// TIA Portal V17 export
// export: Created 2022-07-20T07:01:28.0294157Z, ExportSetting WithDefaults, DisplayName Totally Integrated Automation Portal, DisplayVersion V17, DisplayName TIA Portal Openness, DisplayVersion V17, DisplayName TIA Portal Version Control Interface, DisplayVersion V17, DisplayName SINAMICS Startdrive Advanced, DisplayVersion V17, DisplayName SINAMICS Startdrive G130, G150, S120, S150, SINAMICS MV, S210, DisplayVersion V17, DisplayName SINAMICS Startdrive G110M, G120, G120C, G120D, G120P, G115D, DisplayVersion V17, DisplayName STEP 7 Professional, DisplayVersion V17, DisplayName STEP 7 Safety, DisplayVersion V17, DisplayName WinCC Advanced, DisplayVersion V17
FUNCTION_BLOCK "FB10180_ChucksManager"   // FB10180, LAD
{ S7_Optimized_Access := 'TRUE' }
VERSION : 0.1
// stored: AutoNumber false, IsIECCheckEnabled false, IsRetainMemResEnabled false, MemoryReserve 100, SetENOAutomatically false, UDAEnableTagReadback false
   VAR_INPUT
      ChucksCommunicationIn : Array[0..15] of "stChuckCommunicationIn";
      ChucksParameters : Array[0..15] of "stChuckParameters";
      NumberOfChucks : USInt;
   END_VAR
   VAR_OUTPUT
      ChucksCommunicationOut : Array[0..15] of "stChuckCommunicationOut";
      ChucksSafetyFeedbackHighSignal : Bool;
      ChucksSafetyFeedbackLowSignal : Bool;
      ChucksStartElec : Bool;
      ChucksStopInProgress : Bool;
      ChucksNormalStopDone : Bool;
      ChucksQuickStopDone : Bool;
   END_VAR
   VAR_IN_OUT
      ChucksRequests : Array[0..15] of "stChuckRequests";
      RequestChucksStartElecPulse : Bool;
      RequestChucksStartElecLevel : Bool;
      RequestNormalStop : Bool;
      RequestQuickStop : Bool;
      RequestStartJog : Bool;
      RequestStopJog : Bool;
      ChucksStates : Array[0..15] of "stChuckStates";
   END_VAR
   VAR
      ChucksSameOmacMode : Bool;
      ChucksSameOmacState : Bool;
      ChucksSameMaintenanceFeedback : Bool;
      i : USInt;
      JogManagementStateDiagram : Int;
      R_TRIG_ChucksRequest { S7_SetPoint := 'True'} : R_TRIG;
      R_TRIG_RequestAcknowledge { S7_SetPoint := 'True'} : R_TRIG;
      R_TRIG_ChucksStartElecPulse { S7_SetPoint := 'True'} : R_TRIG;
      R_TRIG_ChucksStartElecLevel { S7_SetPoint := 'True'} : R_TRIG;
      R_TRIG_ErrorOnChucks { S7_SetPoint := 'True'} : R_TRIG;
      R_TRIG_RequestStartJog { S7_SetPoint := 'True'} : R_TRIG;
      R_TRIG_RequestStopJog { S7_SetPoint := 'True'} : R_TRIG;
      F_TRIG_ChucksRequest { S7_SetPoint := 'True'} : F_TRIG;
      F_TRIG_ChucksStartElecLevel { S7_SetPoint := 'True'} : F_TRIG;
      TON_RequestDuration { S7_SetPoint := 'True'} : TON_TIME;
      TON_AcknowledgeDuration { S7_SetPoint := 'True'} : TON_TIME;
      TON_ChucksStartElecPulse { S7_SetPoint := 'True'} : TON_TIME;
      ArrayErrorsChucksLog : Array[0..15] of DInt;
      FB10182_ChuckPortionTracking_Instance { S7_SetPoint := 'True'} : Array[0..15] of "FB10182_ChuckPortionTracking";
   END_VAR
   VAR CONSTANT
      WAIT_FOR_JOG_REQUESTS : Int := 0;
      PARAMETER_CHUCKS : Int := 10;
      START_JOG : Int := 20;
      STOP_JOG : Int := 30;
      JOG_MANAGEMENT_DONE : Int := 40;
   END_VAR
BEGIN

REGION Network 1 (SCL): First Scan
   IF "FirstScan" THEN
       FOR #i := 0 TO #NumberOfChucks DO
           #ChucksCommunicationOut[#i].Acknowledge := FALSE;
           #ChucksCommunicationOut[#i].SheetManagement := 0;
           #ChucksCommunicationOut[#i].StartIdle := FALSE;
           #ChucksCommunicationOut[#i].StartInit := FALSE;
           #ChucksCommunicationOut[#i].Stop := FALSE;
       END_FOR;
       #ChucksCommunicationOut[0].MaintenanceFunction := 1;

       #JogManagementStateDiagram := #WAIT_FOR_JOG_REQUESTS;
   END_IF;
END_REGION

REGION Network 2 (SCL): Edge Signals & Timers
   REGION EDGE SIGNALS
       #R_TRIG_ChucksRequest(CLK := #ChucksRequests[0].StartInit OR #ChucksRequests[0].Stop OR #ChucksRequests[0].StartIdle);
       #R_TRIG_ChucksStartElecPulse(CLK := #RequestChucksStartElecPulse);
       #R_TRIG_ChucksStartElecLevel(CLK := #RequestChucksStartElecLevel);
       #R_TRIG_RequestAcknowledge(CLK := #ChucksRequests[0].Acknowledge);
       #R_TRIG_ErrorOnChucks(CLK := #ChucksStates[0].Error = -1);
       #R_TRIG_RequestStartJog(CLK := #RequestStartJog);
       #R_TRIG_RequestStopJog(CLK := #RequestStopJog);

       #F_TRIG_ChucksRequest(CLK := #ChucksRequests[0].StartInit OR #ChucksRequests[0].Stop OR #ChucksRequests[0].StartIdle);
       #F_TRIG_ChucksStartElecLevel(CLK := #RequestChucksStartElecLevel);
   END_REGION

   REGION TIMERS
       #TON_AcknowledgeDuration(IN := #ChucksCommunicationOut[0].Acknowledge,
                                PT := T#500ms);
       #TON_RequestDuration(IN := #ChucksRequests[0].StartInit OR #ChucksRequests[0].Stop OR #ChucksRequests[0].StartIdle,
                            PT := T#2s);
       #TON_ChucksStartElecPulse(IN := #RequestChucksStartElecPulse,
                                 PT := T#200ms);
   END_REGION
END_REGION

REGION Network 3 (SCL): Chucks Commands Management
   REGION START INIT / START IDLE / STOP / LOAD UNLOAD
       FOR #i := 0 TO #NumberOfChucks DO
           #ChucksCommunicationOut[#i].StartInit := #ChucksRequests[#i].StartInit;
           #ChucksCommunicationOut[#i].StartIdle := #ChucksRequests[#i].StartIdle;
           #ChucksCommunicationOut[#i].Stop := #ChucksRequests[#i].Stop;
           #ChucksCommunicationOut[#i].Load_Unload := #ChucksRequests[#i].Load_Unload;
           #ChucksCommunicationOut[#i].SheetManagement := #ChucksRequests[#i].SheetManagement;
       END_FOR;
   END_REGION

   REGION ACKNOWLEDGE
       IF #R_TRIG_RequestAcknowledge.Q THEN
           #ChucksCommunicationOut[0].Acknowledge := TRUE;
       ELSIF #TON_AcknowledgeDuration.Q THEN
           #ChucksCommunicationOut[0].Acknowledge := FALSE;
       END_IF;
   END_REGION

   REGION START ELEC
       //Start Elec Management
       IF #R_TRIG_ChucksStartElecLevel.Q OR #R_TRIG_ChucksStartElecPulse.Q THEN
           #ChucksStartElec := TRUE;
       ELSIF #TON_ChucksStartElecPulse.Q THEN
           #ChucksStartElec := FALSE;
       ELSIF #RequestNormalStop THEN
           IF #ChucksStates[#NumberOfChucks].ActualPosition > 23120.0 OR (#ChucksStates[#NumberOfChucks].ActualVelocity < 5.0 AND #ChucksStates[#NumberOfChucks / 2].ActualVelocity < 5.0) THEN
               #ChucksRequests[0].Stop := TRUE;
               #ChucksStartElec := FALSE;
           END_IF;
       ELSIF #RequestQuickStop THEN
           #ChucksRequests[0].Stop := TRUE;
           #ChucksStartElec := FALSE;
       ELSE
           #ChucksRequests[0].Stop := FALSE;
       END_IF;
   END_REGION

   REGION JOG
       IF #ChucksStates[0].Error <> 0 OR #R_TRIG_RequestStopJog.Q THEN
           #JogManagementStateDiagram := #STOP_JOG;
       END_IF;

       CASE #JogManagementStateDiagram OF
           #WAIT_FOR_JOG_REQUESTS:
               IF #ChucksStates[0].OmacState = "OMAC_STATE_STOPPED" AND #R_TRIG_RequestStartJog.Q THEN
                   #JogManagementStateDiagram := #PARAMETER_CHUCKS;
               END_IF;
           #PARAMETER_CHUCKS:
               //Request For Chucks
               #ChucksCommunicationOut[0].MaintenanceFunction := 2;

               //Condition To Go To Next Step
               IF #ChucksStates[0].MaintenanceFeedback = #ChucksCommunicationOut[0].MaintenanceFunction THEN
                   #JogManagementStateDiagram := #START_JOG;
               END_IF;
           #START_JOG:
               //Request For Chucks
               #ChucksRequests[0].StartInit := TRUE;

               //Condition To Go To Next Step
               IF #R_TRIG_RequestStopJog.Q THEN
                   #ChucksRequests[0].StartInit := FALSE;
                   #JogManagementStateDiagram := #STOP_JOG;
               END_IF;
           #STOP_JOG:
               #ChucksRequests[0].Stop := TRUE;
               #ChucksCommunicationOut[0].MaintenanceFunction := 1;

               IF #ChucksStates[0].OmacState = "OMAC_STATE_STOPPED" AND #ChucksStates[0].MaintenanceFeedback = 1 THEN
                   #ChucksRequests[0].Stop := FALSE;
                   #JogManagementStateDiagram := #JOG_MANAGEMENT_DONE;
               END_IF;
           #JOG_MANAGEMENT_DONE:
               #ChucksRequests[0].StartInit := FALSE;
               #ChucksRequests[0].Stop := FALSE;
               #JogManagementStateDiagram := #WAIT_FOR_JOG_REQUESTS;
       END_CASE;
   END_REGION

   REGION REQUEST PORTION TRACKING
       FOR #i := 1 TO #NumberOfChucks DO
           #ChucksRequests[#i].RequestPortionTracking := #ChucksRequests[0].RequestPortionTracking;
       END_FOR;
   END_REGION
END_REGION

REGION Network 4 (SCL): Chuck Potion Tracking Management
   FOR #i := 1 TO #NumberOfChucks DO
       #FB10182_ChuckPortionTracking_Instance[#i](EnablePortionTracking:=#ChucksRequests[#i].RequestPortionTracking,
                                                  StartPosition:=#ChucksParameters[#i].PortionTracking_StartDistance,
                                                  EndPosition:=#ChucksParameters[#i].PortionTracking_EndDistance,
                                                  ChuckActualPosition := #ChucksStates[#i].ActualPosition,
                                                  EndPositionReached=>#ChucksStates[#i].PortionTrackingDone);
   END_FOR;
END_REGION

REGION Network 5 (SCL): Chucks States Management
   #ChucksSameOmacMode := TRUE;
   #ChucksSafetyFeedbackHighSignal := FALSE;
   #ChucksSameOmacState := TRUE;
   #ChucksSameMaintenanceFeedback := TRUE;
   #ChucksStates[0].Enabled := TRUE;
   #ChucksStates[0].Initialized := TRUE;
   #ChucksStates[0].Prepositioned := TRUE;
   #ChucksStates[0].ChuckAlive := TRUE;
   #ChucksStates[0].OmacMode := 0;
   #ChucksStates[0].OmacState := 0;
   #ChucksStates[0].Error := 0;
   #ChucksStates[0].MaintenanceFeedback := 0;
   #ChucksStates[0].PortionTrackingDone := FALSE;
   #ChucksStates[0].SafetyFeedbackHighSignal := TRUE;
   #ChucksStates[0].SafetyFeedbackLowSignal := TRUE;

   IF #NumberOfChucks = 0 THEN
       #ChucksStates[0].Enabled := FALSE;
       #ChucksStates[0].Initialized := FALSE;
       #ChucksStates[0].Prepositioned := FALSE;
       #ChucksStates[0].SheetIn := FALSE;
       #ChucksStates[0].ChuckAlive := FALSE;
       #ChucksSameOmacMode := FALSE;
       #ChucksSameOmacState := FALSE;
       #ChucksStates[0].OmacMode := 0;
       #ChucksStates[0].OmacState := 0;
       #ChucksStates[0].Error := 0;
       #ChucksStates[0].MaintenanceFeedback := 0;
       #ChucksStates[0].PortionTrackingDone := FALSE;
   ELSIF #NumberOfChucks >= 1 THEN
       REGION CHUCKS STATES MANAGEMENT
           FOR #i := 1 TO #NumberOfChucks DO
               IF #ChucksStates[#i].ActualPosition < 0.0 THEN
                   #ChucksStates[#i].ActualPosition := 0.0;
               ELSIF #ChucksStates[#i].ActualPosition > 50000.0 THEN
                   #ChucksStates[#i].ActualPosition := 50000.0;
               ELSE
                   #ChucksStates[#i].ActualPosition := #ChucksCommunicationIn[#i].ActualPosition;
               END_IF;
               #ChucksStates[#i].ActualVelocity := #ChucksCommunicationIn[#i].ActualVelocity;
               #ChucksStates[#i].ChuckAlive := #ChucksCommunicationIn[#i].ChuckAlive;
               #ChucksStates[#i].Enabled := #ChucksCommunicationIn[#i].Enabled;
               #ChucksStates[#i].Error := #ChucksCommunicationIn[#i].Error;
               #ChucksStates[#i].Initialized := #ChucksCommunicationIn[#i].Initialized;
               #ChucksStates[#i].OmacMode := #ChucksCommunicationIn[#i].OmacMode;
               #ChucksStates[#i].OmacState := #ChucksCommunicationIn[#i].OmacState;
               #ChucksStates[#i].Prepositioned := #ChucksCommunicationIn[#i].Prepositioned;
               #ChucksStates[#i].SheetIn := #ChucksCommunicationIn[#i].SheetIn;
               #ChucksStates[#i].ChuckAlive := #ChucksCommunicationIn[#i].ChuckAlive;
               #ChucksStates[#i].MaintenanceFeedback := #ChucksCommunicationIn[#i].MaintenanceFeedback;
               #ChucksStates[#i].SafetyFeedbackHighSignal := #ChucksCommunicationIn[#i].ElectricalInputs.%X6;
               #ChucksStates[#i].SafetyFeedbackLowSignal := #ChucksCommunicationIn[#i].ElectricalInputs.%X6;
           END_FOR;
       END_REGION

       REGION DETERMINE COMMON STATE OF CHUCKS
           FOR #i := 1 TO #NumberOfChucks DO
               //Chucks Enabled States Management
               #ChucksStates[0].Enabled := #ChucksStates[0].Enabled AND #ChucksStates[#i].Enabled;

               //Chucks Initialzed States Management
               #ChucksStates[0].Initialized := #ChucksStates[0].Initialized AND #ChucksStates[#i].Initialized;

               //Chucks Prepositionned States Management
               #ChucksStates[0].Prepositioned := #ChucksStates[0].Prepositioned AND #ChucksStates[#i].Prepositioned;

               //Chucks Alive States Management
               #ChucksStates[0].ChuckAlive := #ChucksStates[0].ChuckAlive AND #ChucksStates[#i].ChuckAlive;

               //Chucks Safety Feedback Ok Management
               #ChucksStates[0].SafetyFeedbackHighSignal := #ChucksStates[0].SafetyFeedbackHighSignal AND #ChucksStates[#i].SafetyFeedbackHighSignal;

               //Chucks Safety Feedback Nok Management
               #ChucksStates[0].SafetyFeedbackLowSignal := #ChucksStates[0].SafetyFeedbackLowSignal AND NOT(#ChucksStates[#i].SafetyFeedbackLowSignal);
           END_FOR;
           #ChucksSafetyFeedbackHighSignal := #ChucksStates[0].SafetyFeedbackHighSignal;
           #ChucksSafetyFeedbackLowSignal := #ChucksStates[0].SafetyFeedbackLowSignal;

           //Chucks Sheet In Management
           FOR #i := 1 TO #NumberOfChucks DO
               IF #ChucksStates[#i].SheetIn THEN
                   #ChucksStates[0].SheetIn := TRUE;
                   EXIT;
               ELSE
                   #ChucksStates[0].SheetIn := FALSE;
               END_IF;
           END_FOR;

           //Chucks Error Management
           FOR #i := 1 TO #NumberOfChucks DO
               IF #ChucksStates[#i].Error <> 0 AND #ChucksStates[#i].Error <> 80000 THEN
                   #ChucksStates[0].Error := -1;
                   EXIT;
               ELSE
                   #ChucksStates[0].Error := 0;
               END_IF;
           END_FOR;

           //Chucks Omac Mode Management
           IF #NumberOfChucks = 1 THEN
               #ChucksStates[0].OmacMode := #ChucksStates[1].OmacMode;
           ELSIF #NumberOfChucks > 1 THEN
               FOR #i := 1 TO #NumberOfChucks - 1 DO
                   #ChucksSameOmacMode := #ChucksSameOmacMode AND (#ChucksStates[#i].OmacMode = #ChucksStates[#i + 1].OmacMode);
               END_FOR;
               IF #ChucksSameOmacMode THEN
                   #ChucksStates[0].OmacMode := #ChucksStates[1].OmacMode;
               ELSE
                   #ChucksStates[0].OmacMode := 0;
               END_IF;
           END_IF;

           //Chucks Omac State Management
           IF #NumberOfChucks = 1 THEN
               #ChucksStates[0].OmacState := #ChucksStates[1].OmacState;
           ELSIF #NumberOfChucks > 1 THEN
               FOR #i := 1 TO #NumberOfChucks - 1 DO
                   #ChucksSameOmacState := #ChucksSameOmacState AND (#ChucksStates[#i].OmacState = #ChucksStates[#i + 1].OmacState);
               END_FOR;
               IF #ChucksSameOmacState THEN
                   #ChucksStates[0].OmacState := #ChucksStates[1].OmacState;
               ELSE
                   #ChucksStates[0].OmacState := 0;
               END_IF;
           END_IF;

           //Chucks Maintenace Feedback Management
           IF #NumberOfChucks = 1 THEN
               #ChucksStates[0].MaintenanceFeedback := #ChucksStates[1].MaintenanceFeedback;
           ELSIF #NumberOfChucks > 1 THEN
               FOR #i := 1 TO #NumberOfChucks - 1 DO
                   #ChucksSameMaintenanceFeedback := #ChucksSameMaintenanceFeedback AND (#ChucksStates[#i].MaintenanceFeedback = #ChucksStates[#i + 1].MaintenanceFeedback);
               END_FOR;
               IF #ChucksSameMaintenanceFeedback THEN
                   #ChucksStates[0].MaintenanceFeedback := #ChucksStates[1].MaintenanceFeedback;
               ELSE
                   #ChucksStates[0].MaintenanceFeedback := 0;
               END_IF;
           END_IF;

           //Portion Tracking Done State Managment
           IF #NumberOfChucks = 1 THEN
               #ChucksStates[0].PortionTrackingDone := #ChucksStates[1].PortionTrackingDone;
           ELSIF #NumberOfChucks > 1 THEN
               FOR #i := 1 TO #NumberOfChucks - 1 DO
                   IF #ChucksStates[#i].PortionTrackingDone THEN
                       #ChucksStates[0].PortionTrackingDone := TRUE;
                       EXIT;
                   ELSE
                       #ChucksStates[0].PortionTrackingDone := FALSE;
                   END_IF;
               END_FOR;
           END_IF;
       END_REGION
   END_IF;

   //Logging errors on chucks
   IF #R_TRIG_ErrorOnChucks.Q THEN
       FOR #i := 0 TO 11 DO
           #ArrayErrorsChucksLog[#i] := #ChucksStates[#i].Error;
       END_FOR;
   END_IF;
END_REGION
END_FUNCTION_BLOCK
